Omron CX-Programmer project NuevoProyecto (CX-Programmer 9.61)

# PLC P2E1V2: CJ2M CPU11

## Program NuevoPrograma1 (cyclic task 0)
Local symbols
Amarillo1 1.01 BOOL  ; 1.01
Amarillo2 1.09 BOOL  ; 1.09
Entrada1 0.00 BOOL  ; 0.00
Entrada2 0.01 BOOL  ; 0.01
P0 2.00 BOOL  ; 2.0
P1 2.01 BOOL  ; 2.01
P2 2.02 BOOL  ; 2.02
P3 2.03 BOOL  ; 2.03
P4 2.04 BOOL  ; 2.04
P5 2.05 BOOL  ; 2.05
P6 2.06 BOOL  ; 2.06
P7 2.07 BOOL  ; 2.07
P8 2.08 BOOL  ; 2.08
P9 2.09 BOOL  ; 2.09
Rojo1 1.00 BOOL  ; 1.00
Rojo2 1.08 BOOL  ; 1.08
Verde1 1.02 BOOL  ; 1.02
Verde2 1.10 BOOL  ; 1.10

### Section Sección1
; rung 0
; cells of this rung as drawn
  row 0 col 6: TIM 0000 #300
  vertical links (row, left of col): 
; rung 1
; cells of this rung as drawn
  row 0 col 6: TIM 0001 #50
  vertical links (row, left of col): 
; rung 2
; cells of this rung as drawn
  row 0 col 6: TIM 0002 #200
  vertical links (row, left of col): 
; rung 3
; cells of this rung as drawn
  row 0 col 6: TIM 0003 #50
  vertical links (row, left of col): 
; rung 4
; cells of this rung as drawn
  row 0 col 6: TIM 0004 #10
  vertical links (row, left of col): 
; rung 5
; cells of this rung as drawn
  row 0 col 6: TIM 0005 #10
  vertical links (row, left of col): 
; rung 6
; cells of this rung as drawn
  row 0 col 6: TIM 0006 #300
  vertical links (row, left of col): 
; rung 7
; cells of this rung as drawn
  row 0 col 6: TIM 0007 #10
  vertical links (row, left of col): 
; rung 8
; cells of this rung as drawn
  row 0 col 6: TIM 0008 #10
  vertical links (row, left of col): 

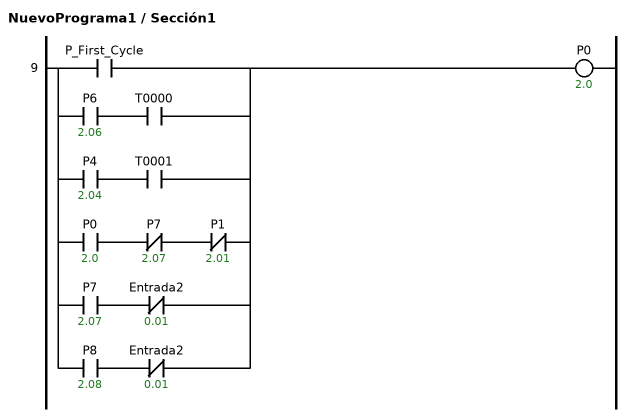
; rung 9
LD P_First_Cycle
LD P6  ; 2.06
AND T0000
ORLD
LD P4  ; 2.04
AND T0001
ORLD
LD P0  ; 2.0
ANDNOT P7  ; 2.07
ANDNOT P1  ; 2.01
ORLD
LD P7  ; 2.07
ANDNOT Entrada2  ; 0.01
ORLD
LD P8  ; 2.08
ANDNOT Entrada2  ; 0.01
ORLD
OUT P0  ; 2.0

### Section END
; rung 0
END(001)